(* Logix 5000 project; controller AdvManLab vendor 1 type 14 code 158 rev 28.12; software revision 28.01; part 5 of 13 *)
(* tags used below, declared in another part *)
   Inp : P_PF52x_Inp;   // Common part of PF523 / PF525 Input Assembly
   Out : P_PF52x_Out;   // Common part of PF523 / PF525 Output Assembly
   Ref_FaultCodeList : P_DescList[1];   // Tag containing List of Fault Codes (DINT) and their Descriptions (STRING)
   Inp_IOFault : BOOL;   // Input Communication Status 0=OK, 1=fail
   Inp_Sim : BOOL;   // 1=Simulate working drive; 0=Start/Stop/ Monitor actual drive
   Inp_OvrdCmd : SINT;   // Override Mode Command: 0=None, 1=Stop, 2=Start Fwd 3=Start Rev
   Cfg_HasJog : BOOL;   // 1=Drive Jog Command enabled/visible, 0=Drive Jog Command not allowed
   Cfg_SetTrack : BOOL;   // 1=PSets track OSets in Oper, OSets track PSets in Prog, 0=no tracking
   Cfg_SetTrackOvrdHand : BOOL;   // 1=Prog/Oper Settings track Override/Hand speed reference
   Cfg_PCmdClear : ALIAS FOR Mode.Cfg_PCmdClear;
   Cfg_OperStopPrio : BOOL;   // 1=OCmd_Stop has priority, accepted any time, 0=OCmd_Stop only in Oper, Maint Mode.
   Cfg_ShedOnFailToStart : BOOL;   // 1=Stop Motor and Alarm on Fail to Start; 0=Alarm only on Fail to Start
   Cfg_MinSpdRef : REAL;   // Minimum Speed Reference in EU (for limiting)
   Cfg_MaxSpdRef : REAL;   // Maximum Speed Reference in EU (for limiting)
   Cfg_SpeedRefRawMin : INT;   // Speed Reference Minimum in Drive (raw) Units (for scaling)
   Cfg_SpeedRefRawMax : INT;   // Speed Reference Maximum in Drive (raw) Units (for scaling)
   Cfg_SpeedRefEUMin : REAL;   // Speed Reference Minimum in Engineering Units (for scaling)
   Cfg_SpeedRefEUMax : REAL;   // Speed Reference Maximum in Engineering Units (for scaling)
   Cfg_OperKeep : SINT;   // Oper keeps control in Prog Mode: .0=Reference, .1=Start/Stop, .2=Fwd/Rev
   Cfg_ProgKeep : SINT;   // Prog keeps control in Oper Mode: .0=Reference, .1=Start/Stop, .2=Fwd/Rev
   PSet_SpeedRef : REAL;   // Program Setting of Speed Reference (EU)
   OSet_SpeedRef : REAL;   // Operator Setting of Speed Reference (EU)
   PCmd_Start : BOOL;   // Program Command to Start Drive
   PCmd_Stop : BOOL;   // Program Command to Stop Drive
   OCmd_Stop : BOOL;   // Operator Command to Stop Drive
   Val_SpeedRef : REAL;   // Speed Reference (target) to drive
   Val_SpeedRefRaw : REAL;   // Copy of Speed Reference Output (in Raw units) for faceplate
   Val_SpeedFdbkRaw : REAL;   // Copy of Speed Feedback Input (in Raw units) for faceplate
   Val_LastFaultCode : DINT;   // Last drive fault code (enum) (Par 951)
   Val_OutCurrent : REAL;   // Drive output current (Amps)
   Val_OutPower : REAL;   // Drive output power (kW)
   SrcQ_IO : SINT;   // Source and Quality of primary I/O (enumeration)
   SrcQ : SINT;   // Source and Quality of primary Val/Sts (enumeration)
   Val_Cmd : SINT;   // Device Command 0=None, 1=Stop, 2=StartFwd 3=StartRev 4=JogFwd 5=JogRev
   Val_Sts : SINT;   // Device Confirmed Sts 0? 1=Stop 2=RunF 3=RunR 4=JogF 5=JogR 6=Stopping 7=Starting F 8=Starting R, 33=Disabled
   Val_Fault : SINT;   // Device Fault Status 0=None, 16=Fail to Start, 17 = Fail to Stop, 18=Drive Fault, 32=I/O Fault, 34=Config Error
   Val_Notify : SINT;   // Current Alarm Level and Acknowledgement (enumeration)
   Sts_Stopped : BOOL;   // 1=Drive requested to stop and is confirmed stopped
   Sts_Starting : BOOL;   // 1=Drive requested to run and awaiting run feedback
   Sts_Running : BOOL;   // 1=Drive requested to run and is confirmed running
   Sts_Stopping : BOOL;   // 1=Drive requested to stop and awaiting stopped feedback
   Sts_Jogging : BOOL;   // 1=Drive requested to Jog
   Sts_CommandDir : BOOL;   // 1=Drive commanded to Forward, 0=Reverse
   Sts_ActualDir : BOOL;   // 1=Drive Actual direction is Forward, 0=Reverse
   Sts_SpeedLimited : BOOL;   // 1=Speed Reference Setting exceeds configured Max/Min limit
   Sts_DigIn1 : BOOL;   // Drive Digital Input 1 Status
   Sts_DigIn2 : BOOL;   // Drive Digital Input 2 Status
   Sts_DigIn3 : BOOL;   // Drive Digital Input 3 Status
   Sts_DigIn4 : BOOL;   // Drive Digital Input 4 Status
   Sts_Disabled : BOOL;   // 1=Drive is Disabled
   Sts_NotRdy : BOOL;   // 1=Motor is Not Ready to Run (independent of Mode)
   Nrdy_OperPrio : BOOL;   // 1=Device Not Ready: Operator State 0 Priority Command Requires Reset
   Nrdy_Fail : BOOL;   // 1=Device Not Ready: Device Failure (Shed Requires Reset)
   Nrdy_IOFault : BOOL;   // 1=Device Not Ready: I/O Fault (Shed Requires Reset)
   Nrdy_Trip : BOOL;   // 1=Device not Ready: Deivce Tripped (Drive Fault)
   Sts_AlmInh : BOOL;   // 1=An Alarm is Shelved, Disabled or Suppressed, display icon
   Sts_Err : BOOL;   // 1=Error in Config: see detail bits for reason
   Err_FdbkRaw : BOOL;   // 1=Erron in Config: Speed Fdbk Raw Min = Max
   Err_FdbkEU : BOOL;   // 1=Error in Config: Speed Fdbk EU Min = Max
   Err_RefEU : BOOL;   // 1=Error in Config: Speed Ref EU Min = Max
   Sts_Hand : ALIAS FOR Mode.Sts_Hand;
   Sts_Maint : ALIAS FOR Mode.Sts_Maint;
   Sts_Ovrd : ALIAS FOR Mode.Sts_Ovrd;
   Sts_Prog : ALIAS FOR Mode.Sts_Prog;
   Sts_Oper : ALIAS FOR Mode.Sts_Oper;
   Sts_FailToStart : ALIAS FOR FailToStart.Inp;   // 1=Drive Failed to Start (One-Shot)
   Sts_FailToStop : ALIAS FOR FailToStop.Inp;   // 1=Drive Failed to Stop
   Sts_DriveFault : ALIAS FOR DriveFault.Inp;   // 1=Drive Fault (see drive display or manual)
   Sts_IOFault : ALIAS FOR IOFault.Inp;   // I/O Comm Fault Status (0=OK, 1=Bad)
   Rdy_Start : BOOL;   // 1=Ready to receive OCmd_Start (enables HMI button)
   Rdy_Stop : BOOL;   // 1=Ready to receive OCmd_Stop (enables HMI button)
   Rdy_Jog : BOOL;   // 1=Ready to receive OCmd_Jog (enables HMI button)
   Rdy_Reset : BOOL;   // 1=Ready to receive OCmd_Reset (enables HMI button)
   Rdy_ResetAckAll : BOOL;   // 1=At least one Alarm or latched Shed condition requires Reset or Ack
   P_PF52x : BOOL;   // Unique Parameter Name for auto - discovery
   Mode : P_Mode;   // Drive Mode Selection
   IOFault : P_Alarm;   // I/O Fault Alarm
   IntlkTrip : P_Alarm;   // Interlock Trip Alarm
   FailToStop : P_Alarm;   // Drive Failed to Stop Alarm
   FailToStart : P_Alarm;   // Drive Failed to Start Alarm
   Wrk_Run : BOOL;   // 1=Drive should be "running", 0=should be "stopped"
   Wrk_StartRetrigT : TIMER;   // Time to pulse start output on start command retrigger (Maint)
   Wrk_StopRetrigT : TIMER;   // Time to pulse stop output on stop command retrigger (Maint)
   Wrk_RunFdbk : BOOL;   // Run Feedback based on mode, simulation, etc. 1=running
   Wrk_Notify : DINT;   // Buffer for building Val_Notify
   DriveFault : P_Alarm;   // Drive Faulted Alarm
   Wrk_SpeedRef : REAL;   // Working copy of Speed Reference (for limiting)
   Wrk_Rev : BOOL;   // Working (internal) Direction 1=Reverse 0=Forward (default)
   Wrk_Jog : BOOL;   // 1=Jog Drive, 0=Drive not jogging
   Wrk_StopT : TIMER;   // Stop Check Timer (for Fail to Stop)
   Wrk_StartT : TIMER;   // Start Check Timer (for Fail to Start)
   Wrk_Cmd : SINT;   // Buffer for building Val_Cmd
   Wrk_Sts : SINT;   // Buffer for building Val_Sts
   Wrk_Fault : SINT;   // Buffer for building Val_Fault
   Wrk_Retrigger : BOOL;   // Maint Start issued while running or Stop while stopped
   Wrk_FaultDescFSC : CONTROL;   // FSC control for Fault Code List search
   Val_FaultDesc : STRING_40;   // Description of Drive Fault (given LastFaultCode)
   Wrk_NotRdy : BOOL;   // Not Ready to run drive, assert Out_Stop
   Wrk_SrcQ : SINT;   // Register for building Source / Quality enumeration
   Wrk_NotRdyONS : BOOL;   // Assert Stop on One-Shot of Sts_NotRdy
   ONS : DINT;
   Running : BOOL;
(* P_PF52x, continued *)

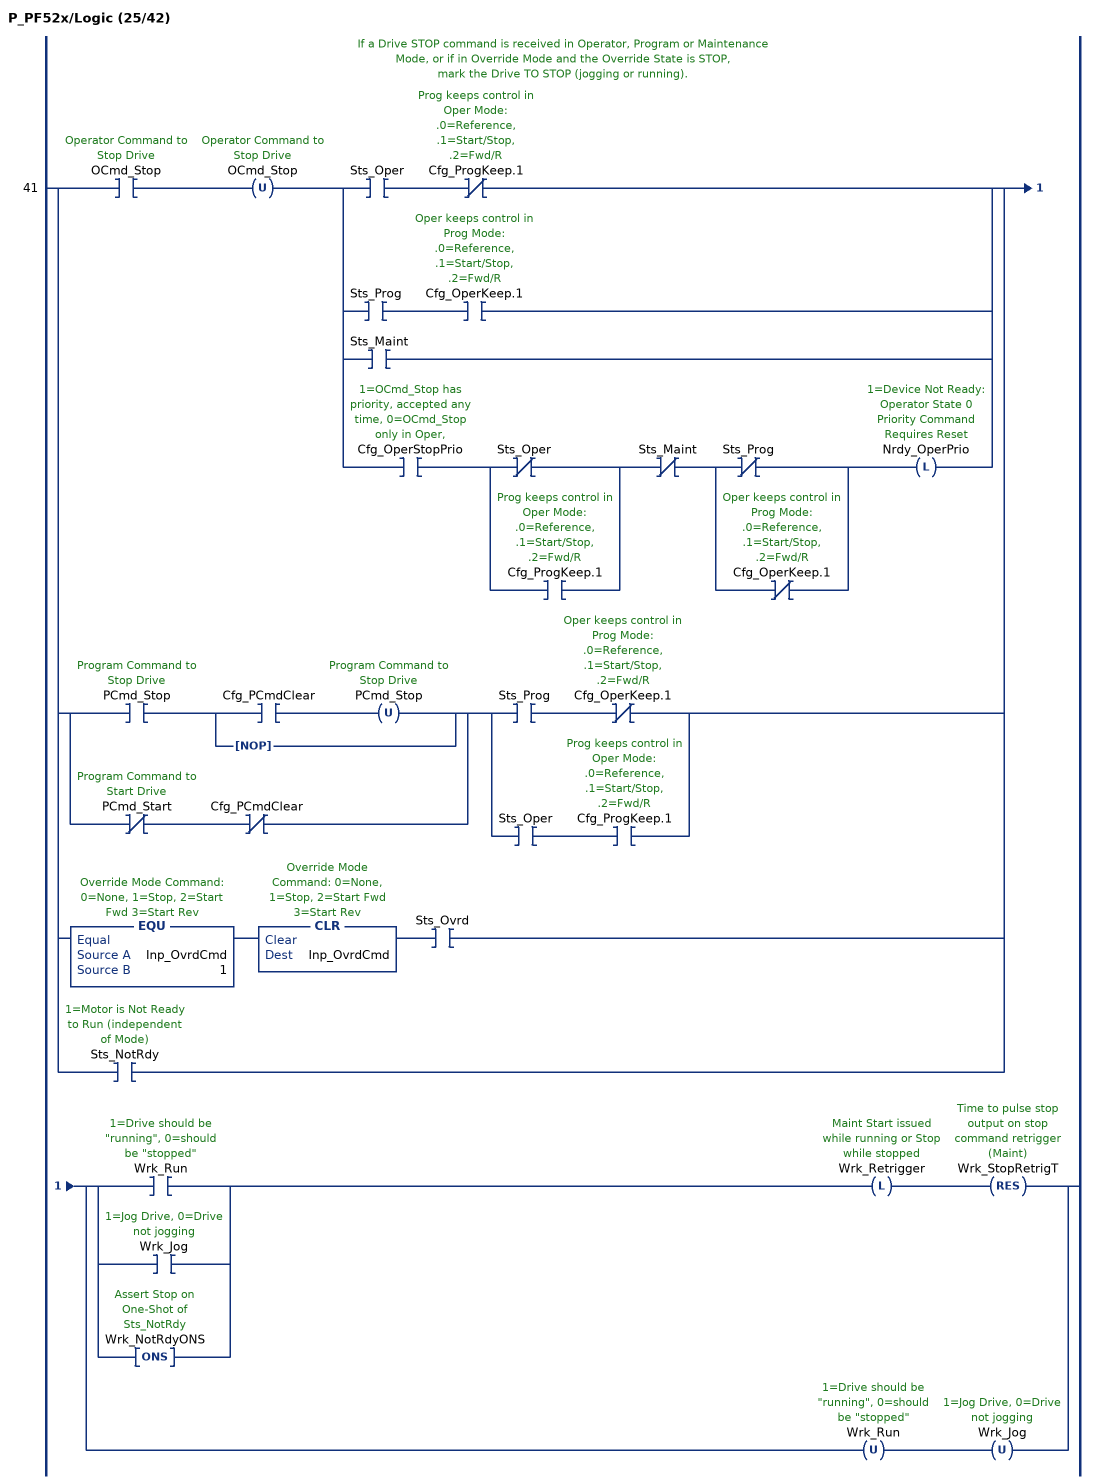
   // If a Drive STOP command is received in Operator, Program or Maintenance
   // Mode, or if in Override Mode and the Override State is STOP,
   // mark the Drive TO STOP (jogging or running).
   41: [XIC(OCmd_Stop) OTU(OCmd_Stop) [XIC(Sts_Oper) XIO(Cfg_ProgKeep.1) ,XIC(Sts_Prog) XIC(Cfg_OperKeep.1) ,XIC(Sts_Maint) ,XIC(Cfg_OperStopPrio) [XIO(Sts_Oper) ,XIC(Cfg_ProgKeep.1) ] XIO(Sts_Maint) [XIO(Sts_Prog) ,XIO(Cfg_OperKeep.1) ] OTL(Nrdy_OperPrio) ] ,[XIC(PCmd_Stop) [XIC(Cfg_PCmdClear) OTU(PCmd_Stop) ,NOP() ] ,XIO(PCmd_Start) XIO(Cfg_PCmdClear) ] [XIC(Sts_Prog) XIO(Cfg_OperKeep.1) ,XIC(Sts_Oper) XIC(Cfg_ProgKeep.1) ] ,EQU(Inp_OvrdCmd,1) CLR(Inp_OvrdCmd) XIC(Sts_Ovrd) ,XIC(Sts_NotRdy) ][[XIC(Wrk_Run) ,XIC(Wrk_Jog) ,ONS(Wrk_NotRdyONS) ] OTL(Wrk_Retrigger) RES(Wrk_StopRetrigT) ,OTU(Wrk_Run) OTU(Wrk_Jog) ];
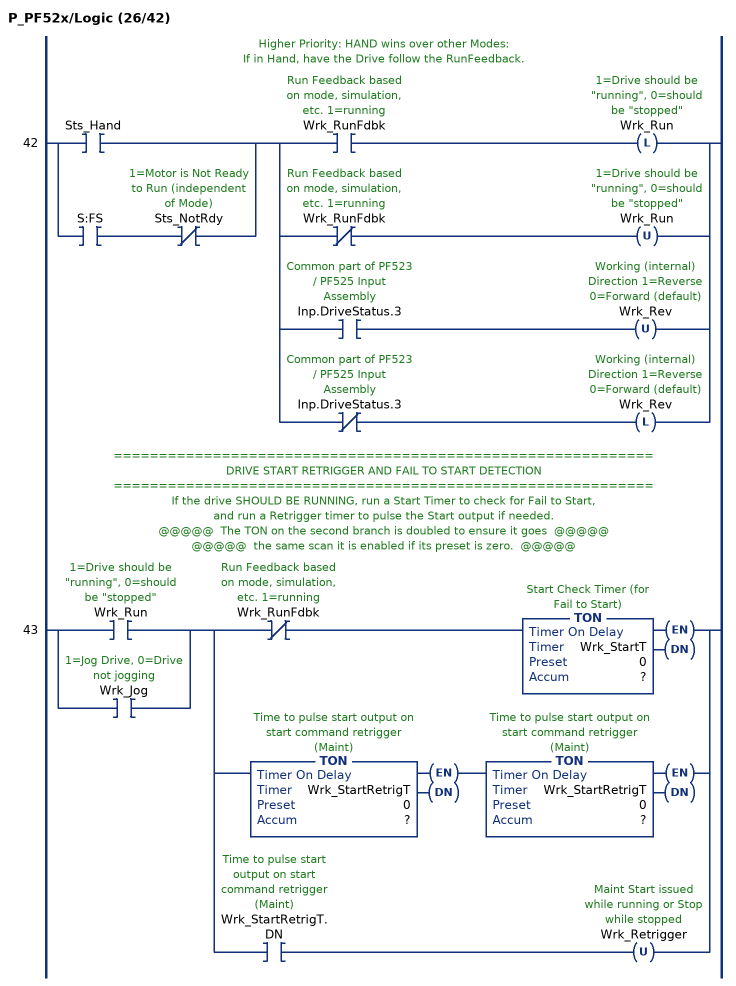
   // Higher Priority: HAND wins over other Modes:
   // If in Hand, have the Drive follow the RunFeedback.
   42: [XIC(Sts_Hand) ,XIC(S:FS) XIO(Sts_NotRdy) ][XIC(Wrk_RunFdbk) OTL(Wrk_Run) ,XIO(Wrk_RunFdbk) OTU(Wrk_Run) ,XIC(Inp.DriveStatus.3) OTU(Wrk_Rev) ,XIO(Inp.DriveStatus.3) OTL(Wrk_Rev) ];
   // ============================================================
   // DRIVE START RETRIGGER AND FAIL TO START DETECTION
   // ============================================================
   // If the drive SHOULD BE RUNNING, run a Start Timer to check for Fail to Start,
   //  and run a Retrigger timer to pulse the Start output if needed.
   // @@@@@  The TON on the second branch is doubled to ensure it goes  @@@@@
   // @@@@@  the same scan it is enabled if its preset is zero.  @@@@@
   43: [XIC(Wrk_Run) ,XIC(Wrk_Jog) ][XIO(Wrk_RunFdbk) TON(Wrk_StartT,?,?) ,TON(Wrk_StartRetrigT,?,?) TON(Wrk_StartRetrigT,?,?) ,XIC(Wrk_StartRetrigT.DN) OTU(Wrk_Retrigger) ];
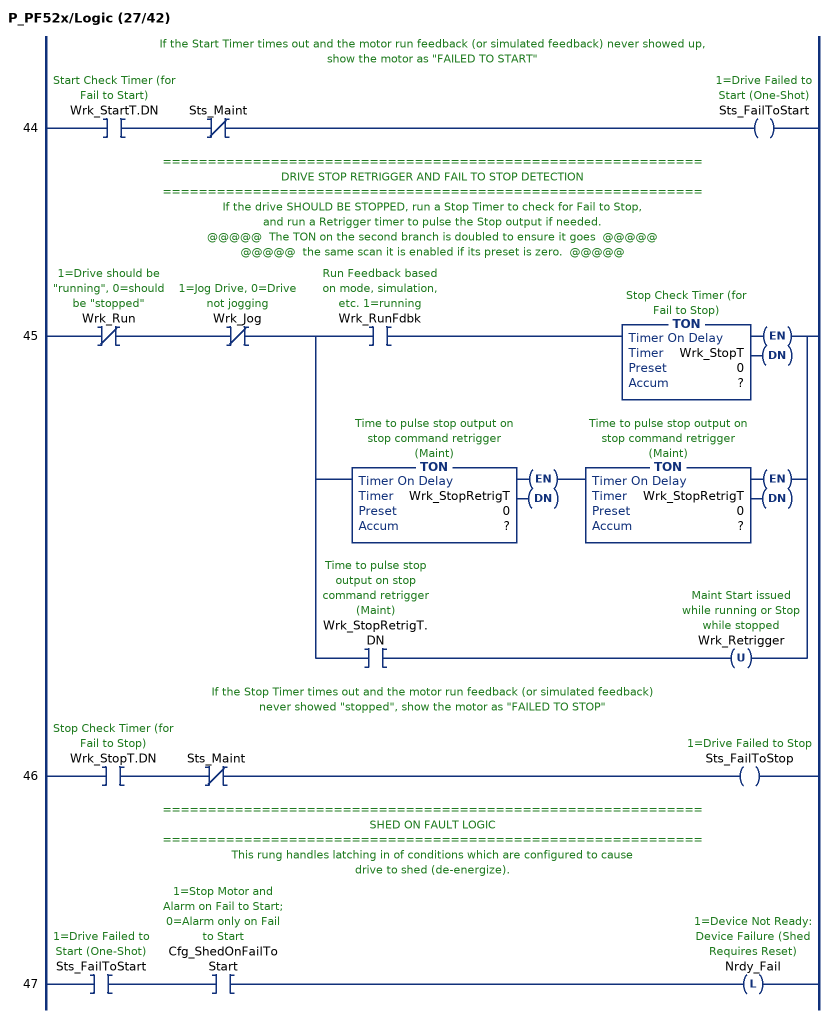
   // If the Start Timer times out and the motor run feedback (or simulated feedback) never showed up,
   // show the motor as "FAILED TO START"
   44: XIC(Wrk_StartT.DN)XIO(Sts_Maint)OTE(Sts_FailToStart);
   // ============================================================
   // DRIVE STOP RETRIGGER AND FAIL TO STOP DETECTION
   // ============================================================
   // If the drive SHOULD BE STOPPED, run a Stop Timer to check for Fail to Stop,
   //  and run a Retrigger timer to pulse the Stop output if needed.
   // @@@@@  The TON on the second branch is doubled to ensure it goes  @@@@@
   // @@@@@  the same scan it is enabled if its preset is zero.  @@@@@
   45: XIO(Wrk_Run)XIO(Wrk_Jog)[XIC(Wrk_RunFdbk) TON(Wrk_StopT,?,?) ,TON(Wrk_StopRetrigT,?,?) TON(Wrk_StopRetrigT,?,?) ,XIC(Wrk_StopRetrigT.DN) OTU(Wrk_Retrigger) ];
   // If the Stop Timer times out and the motor run feedback (or simulated feedback)
   // never showed "stopped", show the motor as "FAILED TO STOP"
   46: XIC(Wrk_StopT.DN)XIO(Sts_Maint)OTE(Sts_FailToStop);
   // ============================================================
   // SHED ON FAULT LOGIC
   // ============================================================
   // This rung handles latching in of conditions which are configured to cause
   // drive to shed (de-energize).
   47: XIC(Sts_FailToStart)XIC(Cfg_ShedOnFailToStart)OTL(Nrdy_Fail);
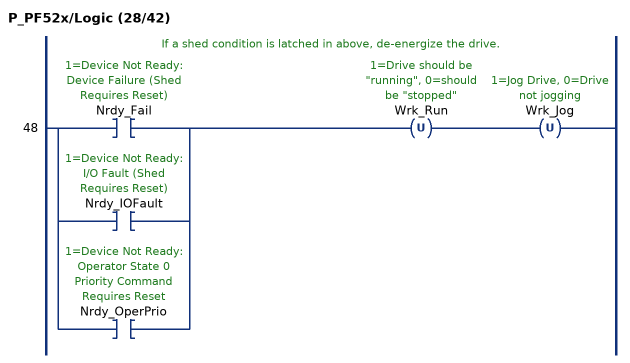
   // If a shed condition is latched in above, de-energize the drive.
   48: [XIC(Nrdy_Fail) ,XIC(Nrdy_IOFault) ,XIC(Nrdy_OperPrio) ]OTU(Wrk_Run)OTU(Wrk_Jog);
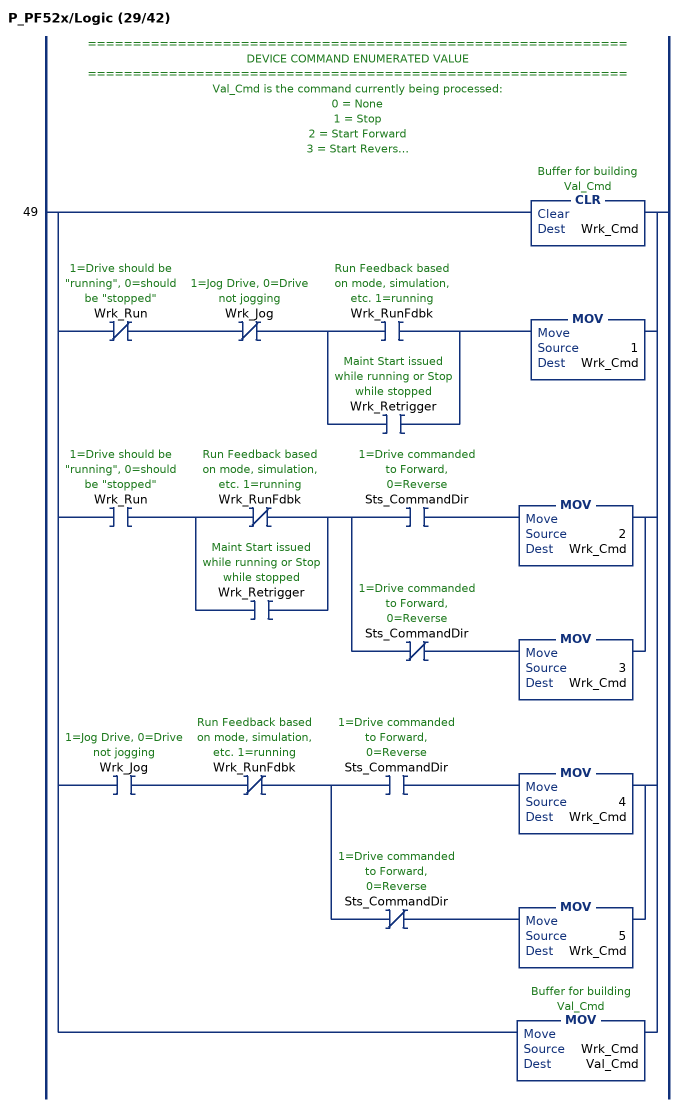
   // ============================================================
   // DEVICE COMMAND ENUMERATED VALUE
   // ============================================================
   // Val_Cmd is the command currently being processed:
   // 0 = None
   // 1 = Stop
   // 2 = Start Forward
   // 3 = Start Reverse
   // 4 = Jog Forward
   // 5 = Jog Reverse
   49: [CLR(Wrk_Cmd) ,XIO(Wrk_Run) XIO(Wrk_Jog) [XIC(Wrk_RunFdbk) ,XIC(Wrk_Retrigger) ] MOV(1,Wrk_Cmd) ,XIC(Wrk_Run) [XIO(Wrk_RunFdbk) ,XIC(Wrk_Retrigger) ] [XIC(Sts_CommandDir) MOV(2,Wrk_Cmd) ,XIO(Sts_CommandDir) MOV(3,Wrk_Cmd) ] ,XIC(Wrk_Jog) XIO(Wrk_RunFdbk) [XIC(Sts_CommandDir) MOV(4,Wrk_Cmd) ,XIO(Sts_CommandDir) MOV(5,Wrk_Cmd) ] ,MOV(Wrk_Cmd,Val_Cmd) ];
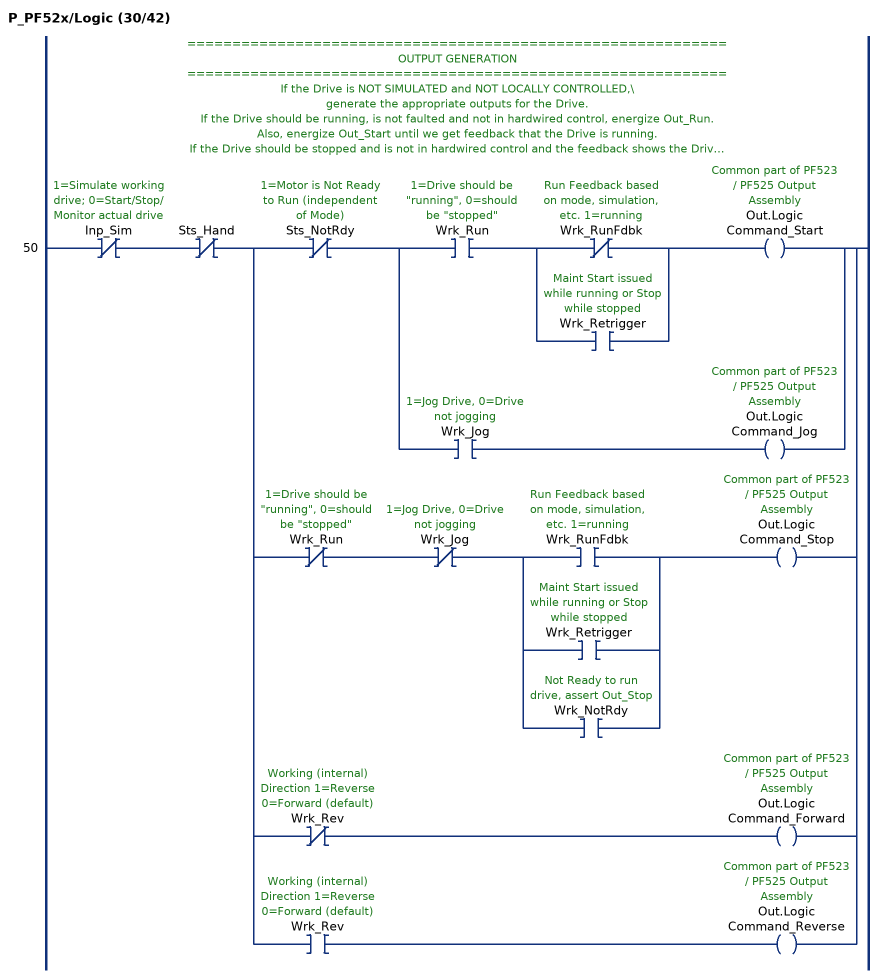
   // ============================================================
   // OUTPUT GENERATION
   // ============================================================
   // If the Drive is NOT SIMULATED and NOT LOCALLY CONTROLLED,\
   // generate the appropriate outputs for the Drive.
   // If the Drive should be running, is not faulted and not in hardwired control, energize Out_Run.
   // Also, energize Out_Start until we get feedback that the Drive is running.
   // If the Drive should be stopped and is not in hardwired control and the feedback shows the Drive
   // is NOT stopped, or if the Drive is Faulted, energize the Out_Stop output to stop the Drive.
   // Finally, if the drive is not simulated, energize the appropriate direction output.
   50: XIO(Inp_Sim)XIO(Sts_Hand)[XIO(Sts_NotRdy) [XIC(Wrk_Run) [XIO(Wrk_RunFdbk) ,XIC(Wrk_Retrigger) ] OTE(Out.LogicCommand_Start) ,XIC(Wrk_Jog) OTE(Out.LogicCommand_Jog) ] ,XIO(Wrk_Run) XIO(Wrk_Jog) [XIC(Wrk_RunFdbk) ,XIC(Wrk_Retrigger) ,XIC(Wrk_NotRdy) ] OTE(Out.LogicCommand_Stop) ,XIO(Wrk_Rev) OTE(Out.LogicCommand_Forward) ,XIC(Wrk_Rev) OTE(Out.LogicCommand_Reverse) ];
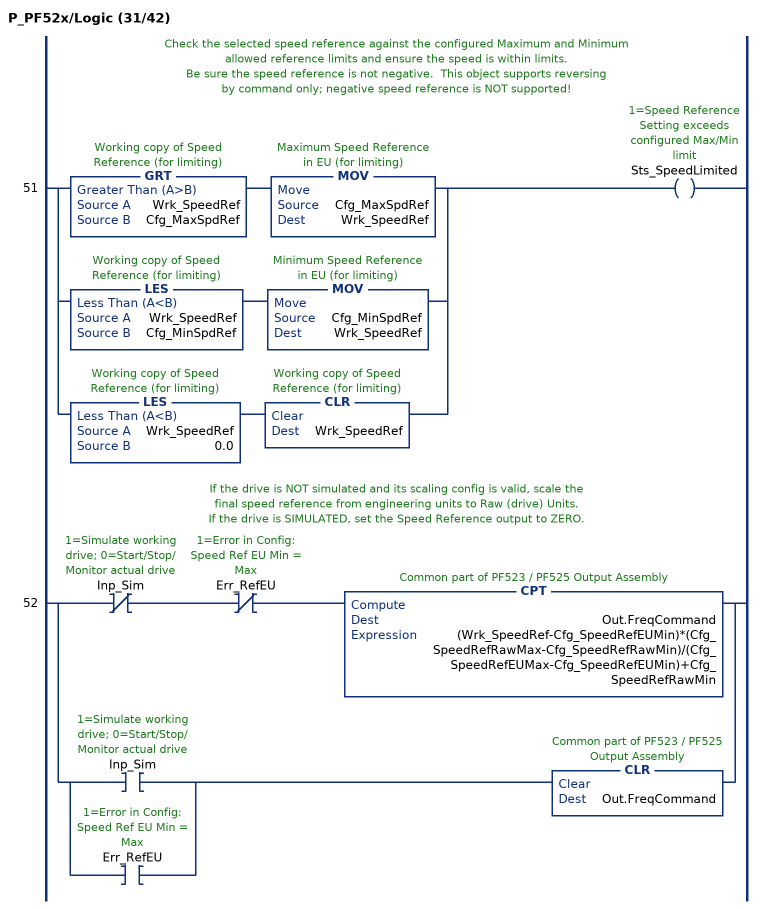
   // Check the selected speed reference against the configured Maximum and Minimum
   // allowed reference limits and ensure the speed is within limits.
   // Be sure the speed reference is not negative.  This object supports reversing
   // by command only; negative speed reference is NOT supported!
   51: [GRT(Wrk_SpeedRef,Cfg_MaxSpdRef) MOV(Cfg_MaxSpdRef,Wrk_SpeedRef) ,LES(Wrk_SpeedRef,Cfg_MinSpdRef) MOV(Cfg_MinSpdRef,Wrk_SpeedRef) ,LES(Wrk_SpeedRef,0.0) CLR(Wrk_SpeedRef) ]OTE(Sts_SpeedLimited);
   // If the drive is NOT simulated and its scaling config is valid, scale the
   // final speed reference from engineering units to Raw (drive) Units.
   // If the drive is SIMULATED, set the Speed Reference output to ZERO.
   52: [XIO(Inp_Sim) XIO(Err_RefEU) CPT(Out.FreqCommand,(Wrk_SpeedRef-Cfg_SpeedRefEUMin)*(Cfg_SpeedRefRawMax-Cfg_SpeedRefRawMin)/(Cfg_SpeedRefEUMax-Cfg_SpeedRefEUMin)+Cfg_SpeedRefRawMin) ,[XIC(Inp_Sim) ,XIC(Err_RefEU) ] CLR(Out.FreqCommand) ];
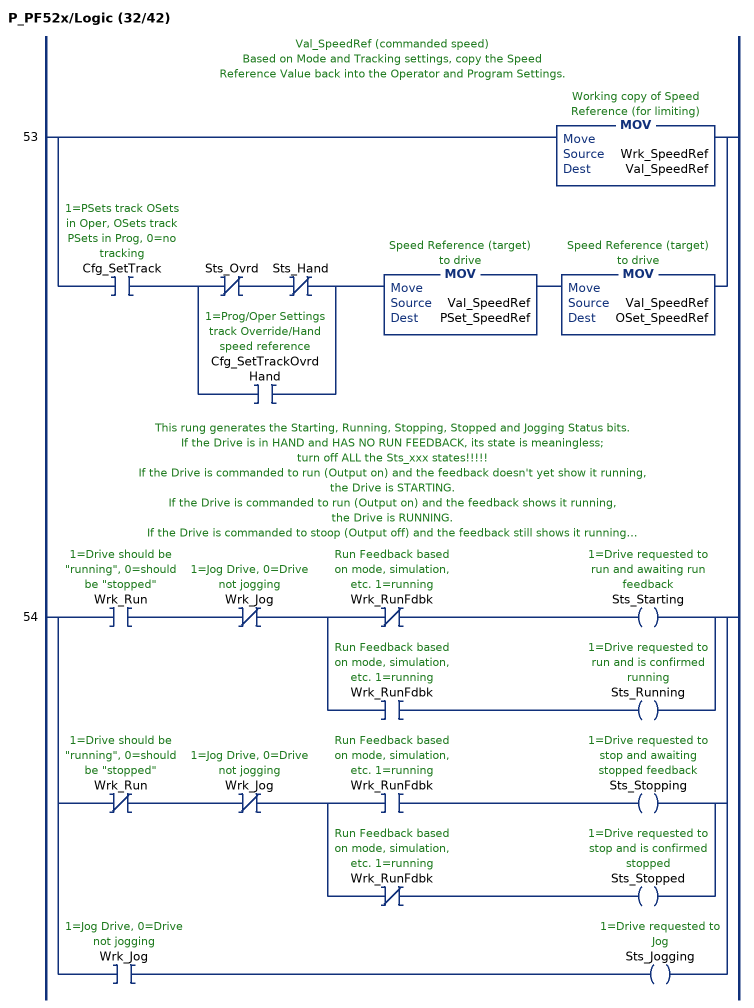
   // Val_SpeedRef (commanded speed)
   // Based on Mode and Tracking settings, copy the Speed
   // Reference Value back into the Operator and Program Settings.
   53: [MOV(Wrk_SpeedRef,Val_SpeedRef) ,XIC(Cfg_SetTrack) [XIO(Sts_Ovrd) XIO(Sts_Hand) ,XIC(Cfg_SetTrackOvrdHand) ] MOV(Val_SpeedRef,PSet_SpeedRef) MOV(Val_SpeedRef,OSet_SpeedRef) ];
   // This rung generates the Starting, Running, Stopping, Stopped and Jogging Status bits.
   // If the Drive is in HAND and HAS NO RUN FEEDBACK, its state is meaningless;
   // turn off ALL the Sts_xxx states!!!!!
   // If the Drive is commanded to run (Output on) and the feedback doesn't yet show it running,
   // the Drive is STARTING.
   // If the Drive is commanded to run (Output on) and the feedback shows it running,
   // the Drive is RUNNING.
   // If the Drive is commanded to stoop (Output off) and the feedback still shows it running,
   // the Drive is STOPPING.
   // If the Drive is commanded to stop (Output off) and the feedback shows it has stopped,
   // the Drive is STOPPED.
   54: [XIC(Wrk_Run) XIO(Wrk_Jog) [XIO(Wrk_RunFdbk) OTE(Sts_Starting) ,XIC(Wrk_RunFdbk) OTE(Sts_Running) ] ,XIO(Wrk_Run) XIO(Wrk_Jog) [XIC(Wrk_RunFdbk) OTE(Sts_Stopping) ,XIO(Wrk_RunFdbk) OTE(Sts_Stopped) ] ,XIC(Wrk_Jog) OTE(Sts_Jogging) ];
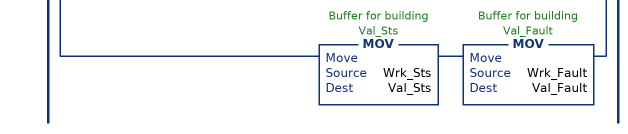
   // Val_Sts is the current device status, as determined by this AOI,
   // based on its knowledge of commands executed and feedback.
   // (This is the status that should be monitored by, for example, FT Historian.)
   // 0 = Powerup / Unknown (Hand Mode with no feedback, for example)
   // 1 = Stopped
   // 2 = Running Forward
   // 3 = Running Reverse
   // 4 = Jogging Forward
   // 5 = Jogging Reverse
   // 6 = Stopping
   // 7 = Starting Forward
   // 8 = Starting Reverse
   // 33 = Device Disabled
   // Val_Fault is the current device fault status, as determined by this AOI,
   // based on its knowledge of commands executed and feedback.
   // (This is the fault status that should be monitored by, for example, FT Historian.)
   // 0 = None
   // 16 = Fail to Start
   // 17 = Fail to Stop
   // 18 = Drive Fault
   // 32 = I/O Fault (from Input)
   // 34 = Configuration Error
   55: [CLR(Wrk_Sts) CLR(Wrk_Fault) ,XIC(Sts_Stopped) MOV(1,Wrk_Sts) ,XIC(Sts_Running) [XIC(Sts_ActualDir) MOV(2,Wrk_Sts) ,XIO(Sts_ActualDir) MOV(3,Wrk_Sts) ] ,XIC(Sts_Jogging) [XIC(Sts_ActualDir) MOV(4,Wrk_Sts) ,XIO(Sts_ActualDir) MOV(5,Wrk_Sts) ] ,XIC(Sts_Stopping) MOV(6,Wrk_Sts) ,XIC(Sts_Starting) [XIC(Sts_CommandDir) MOV(7,Wrk_Sts) ,XIO(Sts_CommandDir) MOV(8,Wrk_Sts) ] ,XIC(Nrdy_Fail) MOV(16,Wrk_Fault) ,XIC(Sts_FailToStop) MOV(17,Wrk_Fault) ,XIC(Sts_DriveFault) MOV(18,Wrk_Fault) ,XIC(Nrdy_IOFault) MOV(32,Wrk_Fault) ,XIC(Sts_Disabled) MOV(33,Wrk_Sts) ,XIC(Sts_Err) MOV(34,Wrk_Fault) ,MOV(Wrk_Sts,Val_Sts) MOV(Wrk_Fault,Val_Fault) ];
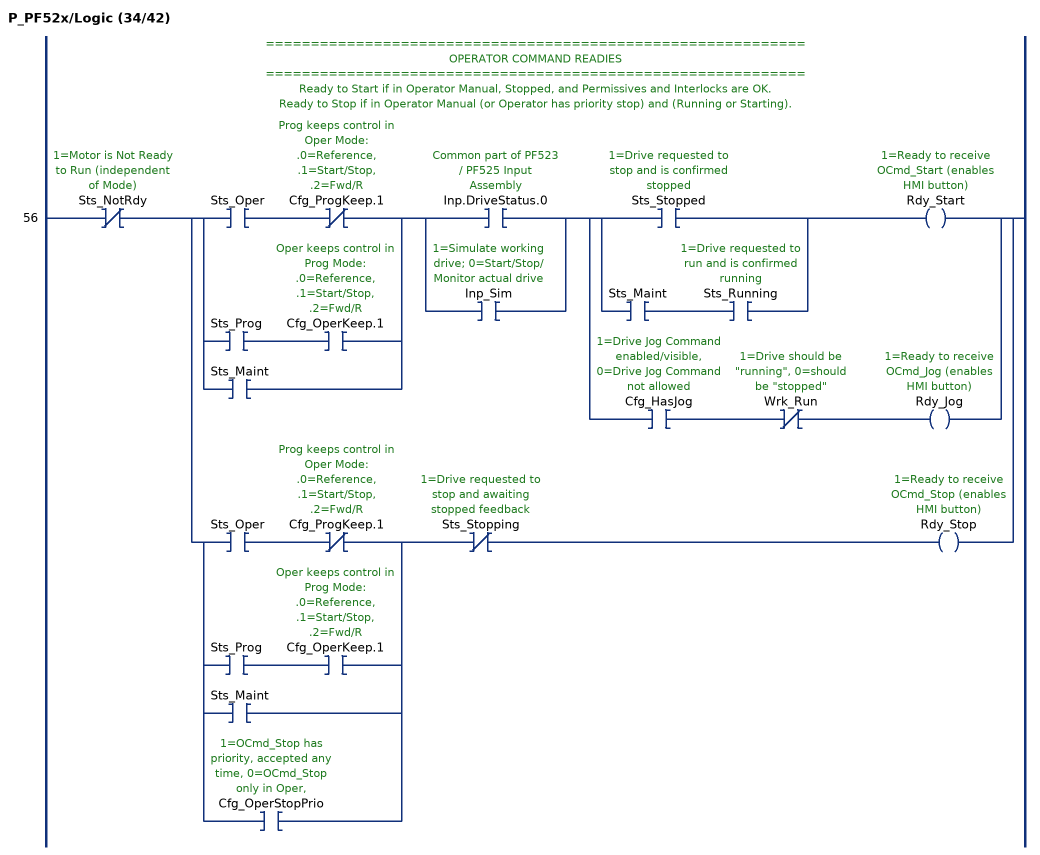
   // ============================================================
   // OPERATOR COMMAND READIES
   // ============================================================
   // Ready to Start if in Operator Manual, Stopped, and Permissives and Interlocks are OK.
   // Ready to Stop if in Operator Manual (or Operator has priority stop) and (Running or Starting).
   56: XIO(Sts_NotRdy)[[XIC(Sts_Oper) XIO(Cfg_ProgKeep.1) ,XIC(Sts_Prog) XIC(Cfg_OperKeep.1) ,XIC(Sts_Maint) ] [XIC(Inp.DriveStatus.0) ,XIC(Inp_Sim) ] [[XIC(Sts_Stopped) ,XIC(Sts_Maint) XIC(Sts_Running) ] OTE(Rdy_Start) ,XIC(Cfg_HasJog) XIO(Wrk_Run) OTE(Rdy_Jog) ] ,[XIC(Sts_Oper) XIO(Cfg_ProgKeep.1) ,XIC(Sts_Prog) XIC(Cfg_OperKeep.1) ,XIC(Sts_Maint) ,XIC(Cfg_OperStopPrio) ] XIO(Sts_Stopping) OTE(Rdy_Stop) ];
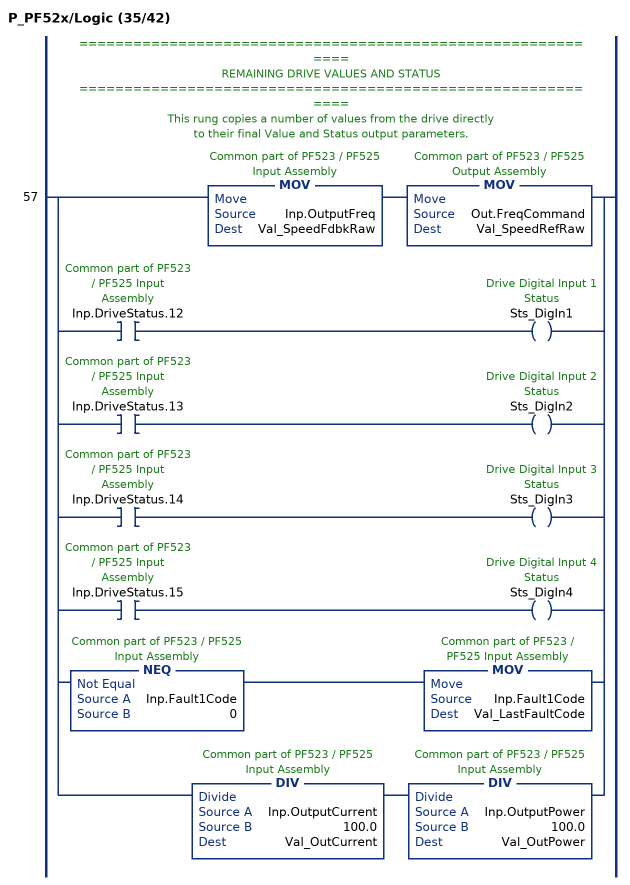
   // ============================================================
   // REMAINING DRIVE VALUES AND STATUS
   // ============================================================
   // This rung copies a number of values from the drive directly
   // to their final Value and Status output parameters.
   57: [MOV(Inp.OutputFreq,Val_SpeedFdbkRaw) MOV(Out.FreqCommand,Val_SpeedRefRaw) ,XIC(Inp.DriveStatus.12) OTE(Sts_DigIn1) ,XIC(Inp.DriveStatus.13) OTE(Sts_DigIn2) ,XIC(Inp.DriveStatus.14) OTE(Sts_DigIn3) ,XIC(Inp.DriveStatus.15) OTE(Sts_DigIn4) ,NEQ(Inp.Fault1Code,0) MOV(Inp.Fault1Code,Val_LastFaultCode) ,DIV(Inp.OutputCurrent,100.0,Val_OutCurrent) DIV(Inp.OutputPower,100.0,Val_OutPower) ];
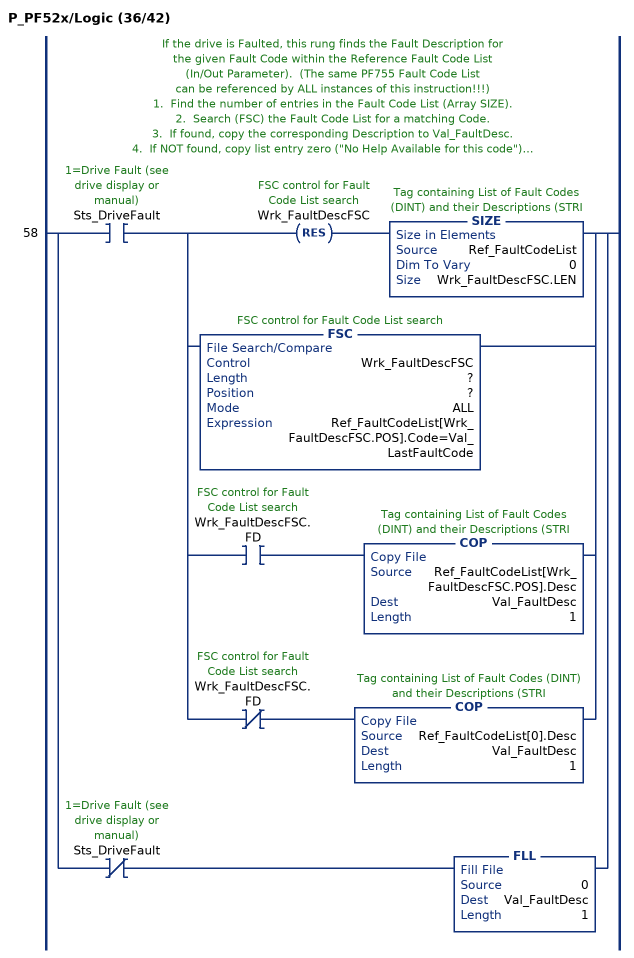
   // If the drive is Faulted, this rung finds the Fault Description for
   // the given Fault Code within the Reference Fault Code List
   // (In/Out Parameter).  (The same PF755 Fault Code List
   // can be referenced by ALL instances of this instruction!!!)
   // 1.  Find the number of entries in the Fault Code List (Array SIZE).
   // 2.  Search (FSC) the Fault Code List for a matching Code.
   // 3.  If found, copy the corresponding Description to Val_FaultDesc.
   // 4.  If NOT found, copy list entry zero ("No Help Available for this code").
   // And if the drive is not faulted, clear the Val_FaultDesc string.
   58: [XIC(Sts_DriveFault) [RES(Wrk_FaultDescFSC) SIZE(Ref_FaultCodeList,0,Wrk_FaultDescFSC.LEN) ,FSC(Wrk_FaultDescFSC,?,?,ALL,Ref_FaultCodeList[Wrk_FaultDescFSC.POS].Code=Val_LastFaultCode) ,XIC(Wrk_FaultDescFSC.FD) COP(Ref_FaultCodeList[Wrk_FaultDescFSC.POS].Desc,Val_FaultDesc,1) ,XIO(Wrk_FaultDescFSC.FD) COP(Ref_FaultCodeList[0].Desc,Val_FaultDesc,1) ] ,XIO(Sts_DriveFault) FLL(0,Val_FaultDesc,1) ];
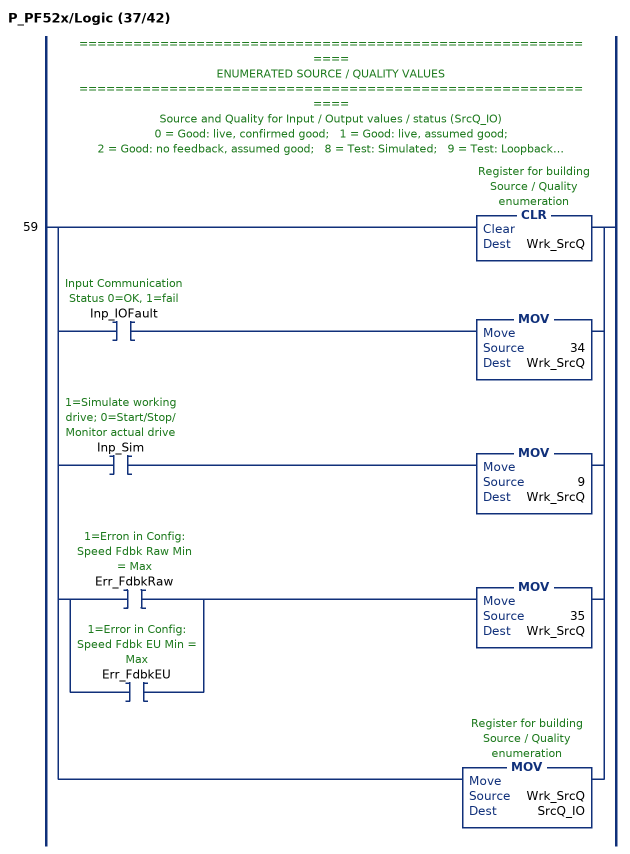
   // ============================================================
   // ENUMERATED SOURCE / QUALITY VALUES
   // ============================================================
   // Source and Quality for Input / Output values / status (SrcQ_IO)
   // 0 = Good: live, confirmed good;   1 = Good: live, assumed good;
   // 2 = Good: no feedback, assumed good;   8 = Test: Simulated;   9 = Test: Loopback;
   // 10 = Test: Manually Entered;   16 = Uncertain: Live, off-spec;
   // 17 = Uncertain, Substituted at Device / Bus;   18 = Uncertain, Substituted at AOI;
   // 19 = Uncertain, using last known good;    20 = Uncertain, using replacement value;
   // 32 = Bad, Signal Failure;   33 = Bad, Channel Fault;
   // 34 = Bad, Module / Comms Fault;   35 = Bad, Invalid Configuration
   59: [CLR(Wrk_SrcQ) ,XIC(Inp_IOFault) MOV(34,Wrk_SrcQ) ,XIC(Inp_Sim) MOV(9,Wrk_SrcQ) ,[XIC(Err_FdbkRaw) ,XIC(Err_FdbkEU) ] MOV(35,Wrk_SrcQ) ,MOV(Wrk_SrcQ,SrcQ_IO) ];
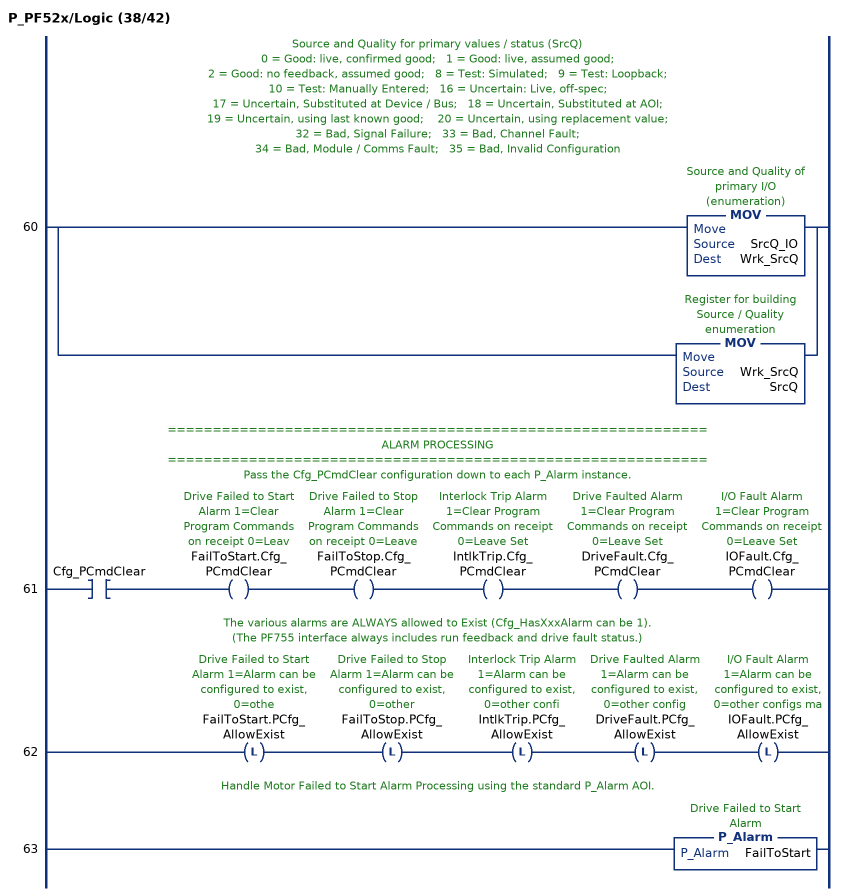
   // Source and Quality for primary values / status (SrcQ)
   // 0 = Good: live, confirmed good;   1 = Good: live, assumed good;
   // 2 = Good: no feedback, assumed good;   8 = Test: Simulated;   9 = Test: Loopback;
   // 10 = Test: Manually Entered;   16 = Uncertain: Live, off-spec;
   // 17 = Uncertain, Substituted at Device / Bus;   18 = Uncertain, Substituted at AOI;
   // 19 = Uncertain, using last known good;    20 = Uncertain, using replacement value;
   // 32 = Bad, Signal Failure;   33 = Bad, Channel Fault;
   // 34 = Bad, Module / Comms Fault;   35 = Bad, Invalid Configuration
   60: [MOV(SrcQ_IO,Wrk_SrcQ) ,MOV(Wrk_SrcQ,SrcQ) ];
   // ============================================================
   // ALARM PROCESSING
   // ============================================================
   // Pass the Cfg_PCmdClear configuration down to each P_Alarm instance.
   61: XIC(Cfg_PCmdClear)OTE(FailToStart.Cfg_PCmdClear)OTE(FailToStop.Cfg_PCmdClear)OTE(IntlkTrip.Cfg_PCmdClear)OTE(DriveFault.Cfg_PCmdClear)OTE(IOFault.Cfg_PCmdClear);
   // The various alarms are ALWAYS allowed to Exist (Cfg_HasXxxAlarm can be 1).
   // (The PF755 interface always includes run feedback and drive fault status.)
   62: OTL(FailToStart.PCfg_AllowExist)OTL(FailToStop.PCfg_AllowExist)OTL(IntlkTrip.PCfg_AllowExist)OTL(DriveFault.PCfg_AllowExist)OTL(IOFault.PCfg_AllowExist);
   // Handle Motor Failed to Start Alarm Processing using the standard P_Alarm AOI.
   63: P_Alarm(FailToStart);
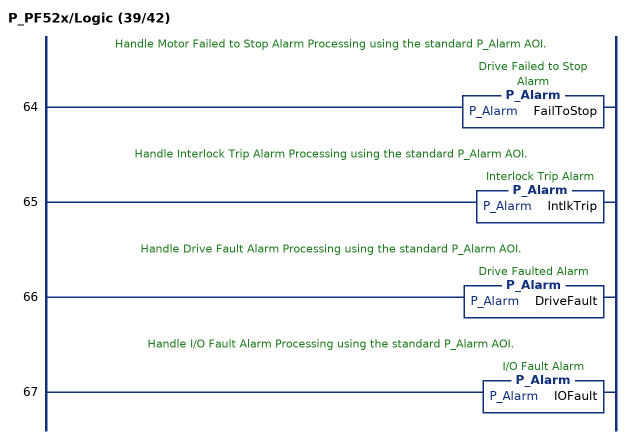
   // Handle Motor Failed to Stop Alarm Processing using the standard P_Alarm AOI.
   64: P_Alarm(FailToStop);
   // Handle Interlock Trip Alarm Processing using the standard P_Alarm AOI.
   65: P_Alarm(IntlkTrip);
   // Handle Drive Fault Alarm Processing using the standard P_Alarm AOI.
   66: P_Alarm(DriveFault);
   // Handle I/O Fault Alarm Processing using the standard P_Alarm AOI.
   67: P_Alarm(IOFault);
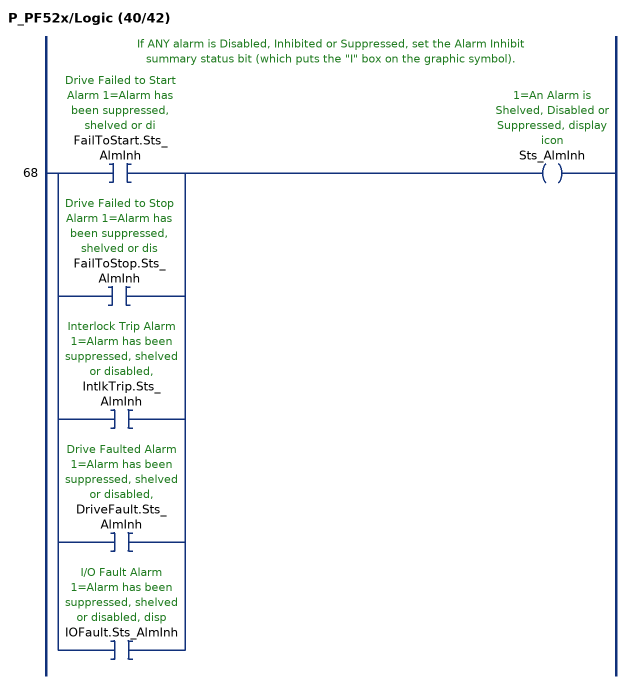
   // If ANY alarm is Disabled, Inhibited or Suppressed, set the Alarm Inhibit
   // summary status bit (which puts the "I" box on the graphic symbol).
   68: [XIC(FailToStart.Sts_AlmInh) ,XIC(FailToStop.Sts_AlmInh) ,XIC(IntlkTrip.Sts_AlmInh) ,XIC(DriveFault.Sts_AlmInh) ,XIC(IOFault.Sts_AlmInh) ]OTE(Sts_AlmInh);
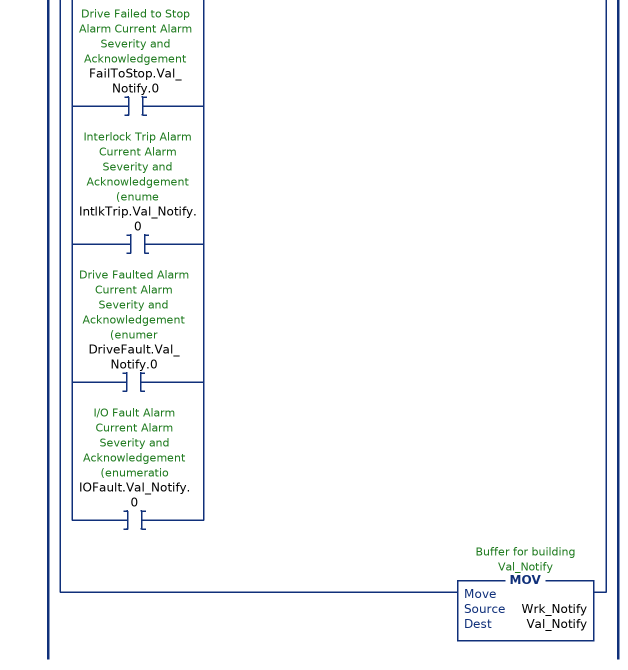
   // ============================================================
   // NOTIFICATION VALUE
   // ============================================================
   // Indicate the current alarm notification level as the max of any of the alarms,
   // and set the low-order bit for reset or ack required:
   // 0 = Not in alarm, acknowledged
   // 1 = Not in alarm, unacknowledged or reset required
   // 2 = Low severity alarm, acknowledged
   // 3 = Low severity alarm, unacknowledged
   // 4 = Medium severity alarm, acknowledged
   // 5 = Medium severity alarm, unacknowledged
   // 6 = High severity alarm, acknowledged
   // 7 = High severity alarm, unacknowledged
   // 8 = Urgent severity alarm, acknowledged
   // 9 = Urgent severity alarm, unacknowledged
   69: [CLR(Wrk_Notify) ,GRT(FailToStart.Val_Notify,Wrk_Notify) MOV(FailToStart.Val_Notify,Wrk_Notify) ,GRT(FailToStop.Val_Notify,Wrk_Notify) MOV(FailToStop.Val_Notify,Wrk_Notify) ,GRT(IntlkTrip.Val_Notify,Wrk_Notify) MOV(IntlkTrip.Val_Notify,Wrk_Notify) ,GRT(DriveFault.Val_Notify,Wrk_Notify) MOV(DriveFault.Val_Notify,Wrk_Notify) ,GRT(IOFault.Val_Notify,Wrk_Notify) MOV(IOFault.Val_Notify,Wrk_Notify) ,[XIC(FailToStart.Val_Notify.0) ,XIC(FailToStop.Val_Notify.0) ,XIC(IntlkTrip.Val_Notify.0) ,XIC(DriveFault.Val_Notify.0) ,XIC(IOFault.Val_Notify.0) ] OTE(Wrk_Notify.0) ,MOV(Wrk_Notify,Val_Notify) ];
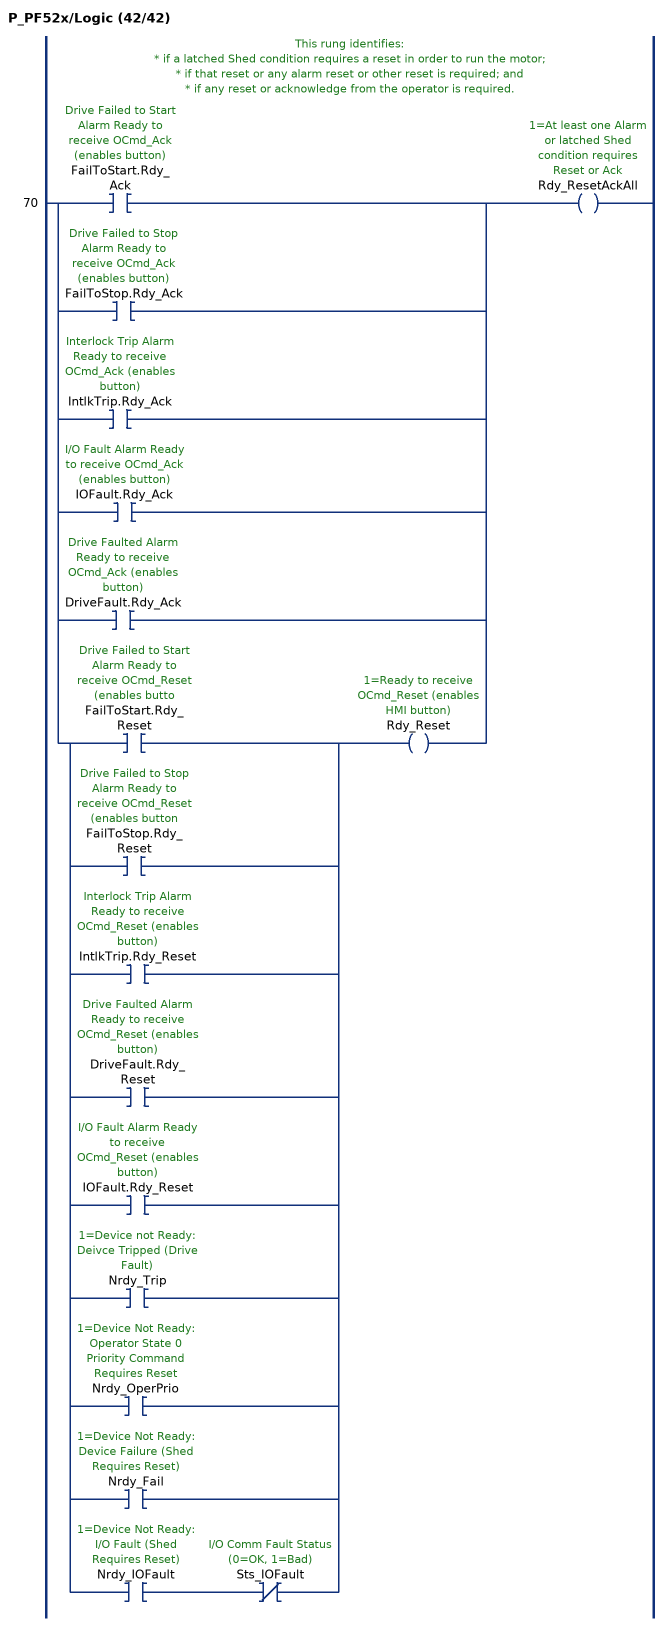
   // This rung identifies:
   // * if a latched Shed condition requires a reset in order to run the motor;
   // * if that reset or any alarm reset or other reset is required; and
   // * if any reset or acknowledge from the operator is required.
   70: [[XIC(FailToStart.Rdy_Ack) ,XIC(FailToStop.Rdy_Ack) ,XIC(IntlkTrip.Rdy_Ack) ,XIC(IOFault.Rdy_Ack) ,XIC(DriveFault.Rdy_Ack) ] ,[XIC(FailToStart.Rdy_Reset) ,XIC(FailToStop.Rdy_Reset) ,XIC(IntlkTrip.Rdy_Reset) ,XIC(DriveFault.Rdy_Reset) ,XIC(IOFault.Rdy_Reset) ,XIC(Nrdy_Trip) ,XIC(Nrdy_OperPrio) ,XIC(Nrdy_Fail) ,XIC(Nrdy_IOFault) XIO(Sts_IOFault) ] OTE(Rdy_Reset) ]OTE(Rdy_ResetAckAll);
END_ROUTINE
